FUNCTION_BLOCK FINAL Profiler
VAR
  dataRef_ : REFERENCE TO ProfilerStruct;
END_VAR

METHOD FB_init : BOOL
VAR_INPUT
	bInitRetains : BOOL; // if TRUE, the retain variables are initialized (warm start / cold start)
	bInCopyCode : BOOL;  // if TRUE, the instance afterwards gets moved into the copy code (online change)
  data : REFERENCE TO ProfilerStruct;
END_VAR
dataRef_ REF= data;
END_METHOD

METHOD popMethod
VAR_INPUT
  hash : UINT; 
END_VAR
IF NOT __ISVALIDREF(dataRef_)
THEN
  RETURN;
END_IF

IF NOT dataRef_.enabled
THEN
  RETURN;
END_IF

dataRef_.depth := dataRef_.depth - 1;
dataRef_.stack[dataRef_.nstack].depth := dataRef_.depth;
dataRef_.stack[dataRef_.nstack].hash := hash;
dataRef_.stack[dataRef_.nstack].starthi := 0;
dataRef_.stack[dataRef_.nstack].startlo := 0;
dataRef_.counter(cpuCntLoDW => dataRef_.stack[dataRef_.nstack].endlo, cpuCntHiDW => dataRef_.stack[dataRef_.nstack].endhi);

IF dataRef_.depth = 0
THEN
  dataRef_.enabled := FALSE;
  dataRef_.stacksize := dataRef_.nstack;
  dataRef_.nstack := 0;
ELSE
  dataRef_.nstack := dataRef_.nstack + 1;  
END_IF
END_METHOD

METHOD pushMethod : BOOL
VAR_INPUT
  hash : UINT;  
END_VAR
IF NOT __ISVALIDREF(dataRef_)
THEN
  RETURN;
END_IF

IF NOT dataRef_.enabled
THEN
  RETURN;
END_IF

dataRef_.stack[dataRef_.nstack].depth := dataRef_.depth;
dataRef_.stack[dataRef_.nstack].hash := hash;
dataRef_.counter(cpuCntLoDW => dataRef_.stack[dataRef_.nstack].startlo, cpuCntHiDW => dataRef_.stack[dataRef_.nstack].starthi);
dataRef_.stack[dataRef_.nstack].endhi := 0;
dataRef_.stack[dataRef_.nstack].endlo := 0;
dataRef_.nstack := dataRef_.nstack + 1;
dataRef_.depth := dataRef_.depth + 1;
END_METHOD

END_FUNCTION_BLOCK

(* stored: Version 1.1.0.1, ProductVersion 3.1.4020.12
   POU Profiler: Id {4c312b8a-7c0e-487b-a95f-8d9579005e8d}, SpecialFunc None
   Method FB_init: Id {abdcc139-61a8-462f-af1e-9d0bfb7f826b}
   Method popMethod: Id {1b9090c0-51e1-4ee1-a2dc-e7ebb71eb6d6}
   Method pushMethod: Id {73ade628-384d-4839-958b-b87e163eaa71} *)
